{attribute 'linkalways'} 
{attribute 'no_explicit_call' := 'This FB is a CLASS and must be accessed using methods or properties'}
{attribute 'enable_dynamic_creation'}
FUNCTION_BLOCK FINAL SQRT_LREAL EXTENDS Node
VAR
	in : _LREAL(0.0);
	out : _LREAL(0.0);
END_VAR

METHOD PUBLIC Clone : I_Node
VAR
	pNode : POINTER TO SQRT_LREAL;
END_VAR
pNode := __NEW(SQRT_LREAL);
Clone := pNode^;
END_METHOD

METHOD FB_init : BOOL
VAR_INPUT
	bInitRetains : BOOL; // if TRUE, the retain variables are initialized (warm start / cold start)
	bInCopyCode : BOOL;  // if TRUE, the instance afterwards gets moved into the copy code (online change)
END_VAR
AddInput('in',THIS^.in);
AddOutput('out', THIS^.out);
END_METHOD

METHOD PROTECTED OnExecute
VAR
END_VAR
out.Value := SQRT(in.Value);
END_METHOD

END_FUNCTION_BLOCK

(* stored: Version 1.1.0.1, ProductVersion 3.1.4024.15
   POU SQRT_LREAL: Id {65dc1e41-6320-497a-8b60-7017b7b75e7b}, SpecialFunc None
   Folder Constructor: Id {1d2b13bb-bf81-460b-896d-c50e7582d185}
   Method Clone: Id {f61b103c-ce93-46b9-8271-2fff65471f71}
   Method FB_init: Id {7c9e600a-9f46-4b7e-9c9b-b01443d7cf69}
   Method OnExecute: Id {387820ec-d91d-4f5f-b900-dc116a99eeba} *)
